// TIA Portal V19 export
DATA_BLOCK "InstLAF_GetSinaEpos"   // DB86
AUTHOR : Siemens Digital Industries
FAMILY : LAF
NAME : LAF_GetSinaEpos
VERSION : 1.1
// stored: InstanceOfName LAF_GetSinaEpos, InstanceOfType FB
"LAF_GetSinaEpos"
   // VAR_INPUT
   //    enable : Bool;
   // END_VAR
   // VAR_OUTPUT
   //    valid { ExternalWritable := 'False'} : Bool;
   //    busy { ExternalWritable := 'False'} : Bool;
   //    error { ExternalWritable := 'False'} : Bool;
   //    status { ExternalWritable := 'False'} : Word;
   //    diagnostics { ExternalWritable := 'False'} : "LAF_typeDiagnostics";
   //    statusWriteRecord { ExternalAccessible := 'False'; ExternalVisible := 'False'; ExternalWritable := 'False'} : DWord;
   //    statusReadRecord { ExternalAccessible := 'False'; ExternalVisible := 'False'; ExternalWritable := 'False'} : DWord;
   // END_VAR
   // VAR_IN_OUT
   //    configuration : Array[*] of "LAF_typeDriveDiagConfig";
   //    moduleInterface : "LAF_typeDriveDiagInterfaceHmi";
   // END_VAR
   // VAR
   //    statInternal { ExternalAccessible := 'False'; ExternalVisible := 'False'; ExternalWritable := 'False'} : Struct
   //       enablePrevious : Bool;
   //       valid : Bool;
   //       busy : Bool;
   //       error : Bool;
   //       errorUserCleared : Bool;
   //       errorAutoCleared : Bool;
   //       disablingCompleted : Bool;
   //       diagnostics : "LAF_typeDiagnostics";
   //       emptyDiagnostics : "LAF_typeDiagnostics";
   //    END_STRUCT;
   //    statMainState { ExternalAccessible := 'False'; ExternalVisible := 'False'; ExternalWritable := 'False'} : DInt;
   //    statArrayMin { ExternalAccessible := 'False'; ExternalVisible := 'False'; ExternalWritable := 'False'} : DInt;
   //    statArrayMax { ExternalAccessible := 'False'; ExternalVisible := 'False'; ExternalWritable := 'False'} : DInt;
   //    instWriteRecord { ExternalAccessible := 'False'; ExternalVisible := 'False'; ExternalWritable := 'False'} : WRREC;
   //    instReadRecord { ExternalAccessible := 'False'; ExternalVisible := 'False'; ExternalWritable := 'False'} : RDREC;
   //    statWriteReq { ExternalAccessible := 'False'; ExternalVisible := 'False'; ExternalWritable := 'False'} : Struct
   //       header : Struct
   //          reqRef : Byte;
   //          reqID : Byte;
   //          axis : Byte;
   //          noPara : Byte;
   //       END_STRUCT;
   //       data : Array[0..235] of Byte;
   //    END_STRUCT;
   //    statReadReq { ExternalAccessible := 'False'; ExternalVisible := 'False'; ExternalWritable := 'False'} : Struct
   //       header : Struct
   //          reqRef : Byte;
   //          reqID : Byte;
   //          axis : Byte;
   //          noPara : Byte;
   //       END_STRUCT;
   //       data : Array[0..235] of Byte;
   //    END_STRUCT;
   //    instActTimer { ExternalAccessible := 'False'; ExternalVisible := 'False'; ExternalWritable := 'False'} : IEC_TIMER;
   //    instReqTimer { ExternalAccessible := 'False'; ExternalVisible := 'False'; ExternalWritable := 'False'} : IEC_TIMER;
   //    statDataTransRun { ExternalAccessible := 'False'; ExternalVisible := 'False'; ExternalWritable := 'False'} : Bool;
   //    statWriteReqSet { ExternalAccessible := 'False'; ExternalVisible := 'False'; ExternalWritable := 'False'} : Bool;
   //    statActTimerIn { ExternalAccessible := 'False'; ExternalVisible := 'False'; ExternalWritable := 'False'} : Bool;
   //    statPrevTimeValue { ExternalAccessible := 'False'; ExternalVisible := 'False'; ExternalWritable := 'False'} : Time;
   //    statActTimerValueAct { ExternalAccessible := 'False'; ExternalVisible := 'False'; ExternalWritable := 'False'} : Time;
   //    statActTimerValueReq { ExternalAccessible := 'False'; ExternalVisible := 'False'; ExternalWritable := 'False'} : Time;
   //    statPrevDriveIndex { ExternalAccessible := 'False'; ExternalVisible := 'False'; ExternalWritable := 'False'} : DInt;
   // END_VAR
BEGIN
END_DATA_BLOCK
